// Mitsubishi GX Works2 project: test   PLC: FX3G

// task Task_01 (event TRUE, interval 0, priority 31): POU_01

PROGRAM POU_01
VAR
  board : ARRAY [0..8] OF INT;
  boardCounter : INT;  (* 棋盤計數器 *)
  boardStack : ARRAY [0..9] OF INT;  (* 移動紀錄 *)
  bestMove : INT;
  randMove : INT;
  winner : INT;
  wstep : INT;  (* 主步數 *)
  ii : INT;
  rand : INT;
  ton1 : TON;
  boardButtonFt : INT;
  flag1 : BOOL;
  temp1 : INT;
END_VAR
(*
名稱：OOXX 挑戰機
版本：v1.0
作者：小麥
*)

(*
M0 - M8 棋盤
M10 開始
M11 先手後手切換
M12 強制結束

D0 - D8 棋盤 
	1 = O
	-1 = X
D9 狀態顯示 (同Y，但只會有正值ABS)
	0 = 預備
	1 = 輪到O
	-1 = 輪到X
	3 = 和局
	4 = O勝
	6 = X勝	
D21 贏的線條
	0 = 空白

D10 難度 (使用 X 有優先權)
	1 = 簡單 X1
	2 = 普通 X2
	3 = 困難 X3
	4 = 極難 X4
*)

(*Debug用 測試段*)
M99 := 
FALSE AND
M10 AND M11 AND M12 AND
M0 AND M1 AND M2 AND
M3 AND M4 AND M5 AND
M6 AND M7 AND M8;

D99 := 
D9 + D10 +
D0 + D1 + D2 +
D3 + D4 + D5 +
D6 + D7 + D8;

(*將遊戲狀態D9轉移至Y*)
ZRST(TRUE, Y0, Y6);
Z2 := ABS(D9);
Y0Z2 := TRUE;

(*開機復歸*)
IF M8002 THEN 
	D8000 := 30000; (*watchdog 時間調整*)
	D10 := 3; (*難度預設 - 困難*)
    wstep := 0;
END_IF;

(*強制結束按扭*)
IF M12 THEN
	M10 := FALSE;
	wstep := 0;
END_IF;

CASE wstep OF
	0:
		(*復歸變數及棋盤*)
		D9 := 0;
		D21 := 0;
		ton1(IN := FALSE);
		boardCounter := 0;
		FOR ii := 0 TO 8 BY 1 DO
			board[ii] := 0;
		END_FOR;
		FOR ii := 0 TO 9 BY 1 DO 
			boardStack[ii] := 0;
		END_FOR;
		M99 := showBoard(TRUE, board);
		
		(*按下開始按鈕*)
		IF M10 THEN 
			IF NOT M11 THEN (*先手後手*)
				D9 := 1;
				wstep := 20;
			ELSE
				D9 := 2;
				wstep := 30;
			END_IF;
		END_IF;
		
	20:
		D9 := getCurrentPlayer(boardCounter);
		
		(*掃描玩家按下的按鈕*)
		FOR ii := 0 TO 8 BY 1 DO 
			Z1 := ii;
			IF M0Z1 AND (board[ii] = 0) THEN (*判斷玩家按鈕 且 該格未被佔用*)
				boardButtonFt := ii;
				wstep := 21;
				RETURN;
			END_IF;
		END_FOR;
	21: (*下緣觸發*)
		Z1 := boardButtonFt;
		IF NOT M0Z1 THEN
			wstep := 22;
		END_IF;
	22: (*下棋*)
		D9 := getCurrentPlayer(boardCounter);
		
		boardStack[boardCounter] := boardButtonFt;
		board[boardButtonFt] := getCurrentPlayer(boardCounter);
		boardCounter := boardCounter + 1;
		M99 := showBoard(TRUE, board); (*顯示棋盤*)
		
		(*輸贏判斷*)
		IF judge(TRUE, board) THEN (*電腦輸*)
			wstep := 40;
			RETURN;
		ELSIF boardCounter = 9 THEN (*和局*)
			wstep := 50;
			RETURN;
		END_IF;
		
		(*產生亂數*)
		rand := LCG((D8013 + 1) * (D8014 + 1)); (*亂數*)
		FOR ii := 0 TO 4 BY 1 DO 
			rand := LCG(rand);
		END_FOR;		
		
		(*X 優先權*)
		FOR ii := 1 TO 4 BY 1 DO 
			temp1 := 4 - ii + 1;
			Z1 := temp1;
			IF X0Z1 THEN
				(*照難度決定使用計算或隨機*)
				CASE temp1 OF
					1: (*100%隨機*)
						wstep := 30;
					2: (*50%隨機*)
						IF (rand MOD 2) = 0 THEN
							wstep := 31;
						ELSE
							wstep := 30;
						END_IF;
					3: (*20%隨機*)
						IF (rand MOD 5) = 0 THEN
							wstep := 31;
						ELSE
							wstep := 30;
						END_IF;
					4: (*0%隨機*)
						wstep := 31;		
				END_CASE;
				
				RETURN; (*下方直接跳過*)
			END_IF;
		END_FOR;
		
		(*照難度決定使用計算或隨機*)
		CASE D10 OF
			1: (*100%隨機*)
				wstep := 30;
			2: (*50%隨機*)
				IF (rand MOD 2) = 0 THEN
					wstep := 31;
				ELSE
					wstep := 30;
				END_IF;
			3: (*20%隨機*)
				IF (rand MOD 5) = 0 THEN
					wstep := 31;
				ELSE
					wstep := 30;
				END_IF;
			4: (*0%隨機*)
				wstep := 31;		
		END_CASE;
		
	30: (*隨機下棋*)
		randMove := randomDraw(TRUE, board);
		boardStack[boardCounter] := randMove;
		board[randMove] := getCurrentPlayer(boardCounter);
		boardCounter := boardCounter + 1;
		M99 := showBoard(TRUE, board); (*顯示棋盤*)
		
		(*輸贏判斷*)
		IF judge(TRUE, board) THEN (*電腦輸*)
			wstep := 40;
		ELSIF boardCounter = 9 THEN (*和局*)
			wstep := 50;
		ELSE (*繼續*)
			wstep := 20;
		END_IF;
	31:
		(*第一層剪枝*)
		IF boardCounter = 1 THEN
			wstep := 32;
			RETURN;
		END_IF;
		(*下棋*)
		bestMove := findBestMove(TRUE, board, boardCounter, boardStack);
		boardStack[boardCounter] := bestMove;
		board[bestMove] := getCurrentPlayer(boardCounter);
		boardCounter := boardCounter + 1;
		M99 := showBoard(TRUE, board); (*顯示棋盤*)
		
		(*輸贏判斷*)
		IF judge(TRUE, board) THEN (*電腦輸*)
			wstep := 40;
		ELSIF boardCounter = 9 THEN (*和局*)
			wstep := 50;
		ELSE (*繼續*)
			wstep := 20;
		END_IF;
	32: (*第一層剪枝*)
		IF board[4] = 1 THEN (*畫中間*)
			(*產生亂數*)
			rand := LCG((D8013 + 1) * (D8014 + 1)); (*亂數*)
			FOR ii := 0 TO 4 BY 1 DO 
				rand := LCG(rand);
			END_FOR;		
			
			IF (rand MOD 2) = 0 THEN
				bestMove := 0;
			END_IF;
			IF (rand MOD 3) = 0 THEN
				bestMove := 2;
			END_IF;
			IF (rand MOD 5) = 0 THEN
				bestMove := 6;
			END_IF;
			IF (rand MOD 7) = 0 THEN
				bestMove := 8;
			END_IF;
		ELSE
			bestMove := 4; 
		END_IF;
		boardStack[boardCounter] := bestMove;
		board[bestMove] := getCurrentPlayer(boardCounter);
		boardCounter := boardCounter + 1;
		M99 := showBoard(TRUE, board); (*顯示棋盤*)
		wstep := 20;
		
	40: (*有勝負*)
		D9 := getCurrentPlayer(boardCounter) + 5;
		
		ton1(IN := TRUE, PT := T#5s);
		IF ton1.Q THEN
			M10 := FALSE;
			wstep := 0;
		END_IF;	
	50: (*和局*)
		D9 := 3;
		
		ton1(IN := TRUE, PT := T#5s);
		IF ton1.Q THEN
			M10 := FALSE;
			wstep := 0;
		END_IF;
END_CASE;
END_PROGRAM

FUNCTION showBoard
VAR_INPUT
  board : ARRAY [0..8] OF INT;  (* 棋盤 *)
  trigger : BOOL;
END_VAR
VAR
  ii : INT;
END_VAR
IF trigger THEN
	FOR ii := 0 TO 8 BY 1 DO
		Z0 := ii;
		D0Z0 := board[ii];
	END_FOR;
END_IF;
END_FUNCTION

FUNCTION judge
VAR
  ii : INT;
  result : BOOL;
END_VAR
VAR_INPUT
  board : ARRAY [0..8] OF INT;  (* 棋盤 *)
  trigger : BOOL;
END_VAR
IF trigger THEN
	D21 := -1;
	result := FALSE;
	
	(*橫*)
	FOR ii := 0 TO 6 BY 3 DO
		IF (board[ii] = board[ii + 1]) AND (board[ii] = board[ii + 2]) AND (board[ii] <> 0) THEN
			D21 := (ii / 3) + 1;
			result := TRUE;
		END_IF;
	END_FOR;
	
	(*直*)
	FOR ii := 0 TO 2 BY 1 DO
		IF (board[ii] = board[ii + 3]) AND (board[ii] = board[ii + 6]) AND (board[ii] <> 0) THEN
			D21 := (3 + ii) + 1;
			result := TRUE;
		END_IF;
	END_FOR;
	
	(*斜*)
	IF (board[0] = board[4]) AND (board[0] = board[8]) AND (board[0] <> 0) THEN
		D21 := 6 + 1;
		result := TRUE;
	END_IF;
	IF (board[2] = board[4]) AND (board[2] = board[6]) AND (board[2] <> 0) THEN
		D21 := 7 + 1;	
		result := TRUE;
	END_IF;	
END_IF;

judge := result;
END_FUNCTION

FUNCTION findBestMove
VAR_INPUT
  trigger : BOOL;
  board : ARRAY [0..8] OF INT;  (* 棋盤 *)
  boardCounter : INT;
  boardStack : ARRAY [0..9] OF INT;  (* 棋盤紀錄 *)
END_VAR
VAR
  result : INT;
  score : INT;
  flag1 : BOOL;
  flag2 : BOOL;
  scoreStack : ARRAY [0..9] OF INT;
  currentPlayer : INT;
  move1 : INT;
  ii : INT;
  Copyboard : ARRAY [0..8] OF INT;
  CopyBoardCounter : INT;
  CopyboardStack : ARRAY [0..9] OF INT;
END_VAR
(*
感謝:
The Coding Train - Coding Challenge 154
	https://bit.ly/3XzAUd0
trincot 於 StackOverflow 提拱技術支援
	https://bit.ly/3GWZInZ
*)

IF trigger THEN
	result := -1;
	
	(*暫存*)
	CopyBoard := board;
	CopyBoardCounter := boardCounter;
	CopyBoardStack := boardStack;
	
	WHILE TRUE DO
		WDT(TRUE); (*防死機*)
	    currentPlayer := getCurrentPlayer(CopyBoardCounter); (*取得當前玩家*)

	    IF judge(TRUE, Copyboard) THEN (*有輸贏*)
	        scoreStack[CopyBoardCounter] := (CopyBoardCounter - 10) * currentPlayer;
	    ELSIF CopyBoardCounter = 9 THEN (*和局*)
	        scoreStack[CopyBoardCounter] := 0;
	    ELSE
	        CopyBoardStack[CopyBoardCounter] := -1;
	        scoreStack[CopyBoardCounter] := currentPlayer * -1 * 10; (*先將未計算的值處理好，方便後面比較*)
	        CopyBoardCounter := CopyBoardCounter + 1;
	    END_IF;
	    
		(*當9個格字都被畫了則跳出*)
	    flag1 := TRUE;
	    WHILE (MOVE1 = 9) OR flag1 DO
			WDT(TRUE); (*防死機*)
	        flag1 := FALSE;
			
			(*該路徑已計算完成*)
	        CopyBoardCounter := CopyBoardCounter - 1;
	        IF CopyBoardCounter < boardCounter THEN
	            EXIT;
	        END_IF;
	
	        MOVE1 := CopyBoardStack[CopyBoardCounter];
	        IF MOVE1 >= 0 THEN
				(*讀取上一次計算的分數*)
	            score := scoreStack[CopyBoardCounter + 1];
	
	            (*對兩者做XNOR，當為 "O" 的時候則越大越好，若為 "X" 則越小越好*)
				IF ((CopyBoard[MOVE1] = 1) = (score >= scoreStack[CopyBoardCounter])) THEN 
	                scoreStack[CopyBoardCounter] := score;
	                
					(*算到最後了，即可計算出最佳解*)
					IF CopyBoardCounter = boardCounter THEN
	                    result := MOVE1;
	                END_IF;
	            END_IF;
	            
	            CopyBoard[MOVE1] := 0;
	        END_IF;
	        
	        (*如果格子已經被畫過了則跳過，直到遇到空格*)
			flag2 := TRUE;
	        WHILE ((CopyBoard[MOVE1] <> 0) AND (MOVE1 < 9)) OR flag2 DO
				WDT(TRUE); (*防死機*)
	            flag2 := FALSE;
	            MOVE1 := MOVE1 + 1;
	        END_WHILE;
	    END_WHILE;
	
	    IF CopyBoardCounter < boardCounter THEN
	        EXIT;
	    END_IF;
	
		(*改變暫存*)
	    CopyBoard[MOVE1] := getCurrentPlayer(CopyBoardCounter);
	    CopyBoardStack[CopyBoardCounter] := MOVE1;
	    CopyBoardCounter := CopyBoardCounter + 1;
	END_WHILE;
END_IF;

findBestMove := result;
END_FUNCTION

FUNCTION randomDraw
VAR_INPUT
  trigger : BOOL;
  board : ARRAY [0..8] OF INT;
END_VAR
VAR
  result : INT;
  ii : INT;
  rand : INT;
END_VAR
IF trigger THEN
	rand := (D8013 + 1) * (D8014 + 1) * (D8019 + 1);
	FOR ii := 0 TO 4 BY 1 DO
		rand := LCG(rand);
	END_FOR;
	
	(*若計算到已被畫過的格子則不停重新計算*)
	WHILE board[rand MOD 9] <> 0 DO 
		rand := LCG(rand);
	END_WHILE;	
END_IF;

RandomDraw := rand MOD 9;
END_FUNCTION

FUNCTION LCG
VAR_INPUT
  seed : INT;
END_VAR
LCG := ABS((6997 * seed + 9851)) MOD 29231;
END_FUNCTION

FUNCTION getCurrentPlayer
VAR_INPUT
  currentPlayer : INT;
END_VAR
(*只會有 1 or -1*)
getCurrentPlayer := 1 - (currentPlayer MOD 2) * 2;
END_FUNCTION
